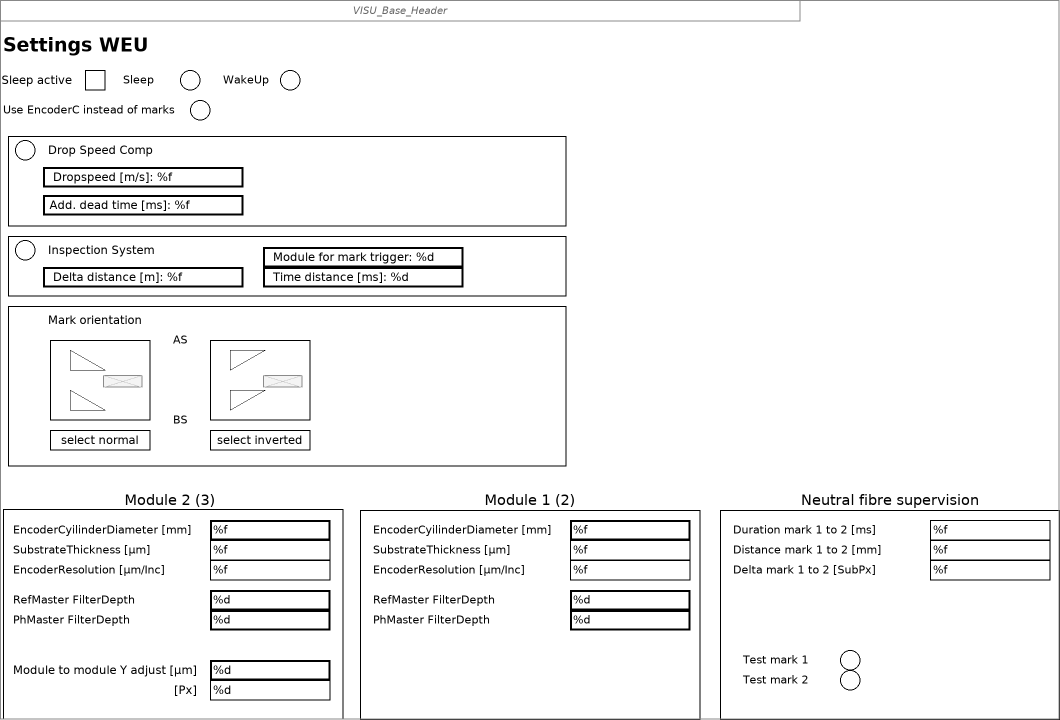
VISUALIZATION VISU_SettingsWeu  // 1060x720
    Rectangle (3,509 340x210)
    Ellipse (190,100 20x20), tooltip "Sim VEncoder"
        toggle PRG_PRINT.bL_EnableEncTrig
    Rectangle (0,100 180x20), "Use EncoderC instead of marks"
    Rectangle (0,30 300x30), "Settings WEU"
    Rectangle (360,510 340x210)
    Label (0,490 340x20), "Module 2 (3)"
    Label (360,490 340x20), "Module 1 (2)"
    Rectangle (10,560 180x20), "EncoderResolution [µm/Inc]"
    Rectangle (210,560 120x20), "%f", text variable: PRG_PRINT.fL_ResolutionEncoder[2]
        OnMouseClick: write the text variable via Default
    Frame (0,0 800x21)
        shows VISU_Base_Header()
    Rectangle (8,136 558x90)
    Ellipse (15,140 20x20), colour toggle: PRG_PRINT.bL_UseSpeedCompensation
        toggle PRG_PRINT.bL_UseSpeedCompensation
    Rectangle (45,140 124x20), "Drop Speed Comp"
    Rectangle (43,167 200x20), "Dropspeed [m/s]: %f", text variable: PRG_PRINT.fL_DropSpeed
        OnMouseDown: write the text variable via Edit
    Rectangle (43,195 200x20), "Add. dead time [ms]: %f", text variable: PRG_PRINT.fL_DropSpeedAddTime
        OnMouseDown: write the text variable via Edit
    Rectangle (370,520 187x20), "EncoderCyilinderDiameter [mm]"
    Rectangle (570,520 120x20), "%f", text variable: PRG_PRINT.lEncoderCylinderDiameter[1]
        OnMouseClick: write the text variable via Default
    RoundedRectangle (85,70 20x20), colour toggle: PRG_MACHINE.sO_SystemCmd.bSleep
    Rectangle (0,70 75x20), "Sleep active"
    Ellipse (180,70 20x20), tooltip "Sim VEncoder"
        tap PRG_MACHINE.bL_SleepVisu
    Rectangle (120,70 55x20), "Sleep"
    Ellipse (280,70 20x20), tooltip "Sim VEncoder"
        tap PRG_MACHINE.bL_WakeUpVisu
    Rectangle (220,70 55x20), "WakeUp"
    Rectangle (210,660 120x20), "%d", text variable: PRG_PRINT.nPrintModuleAdjustY[2]
        OnMouseClick: write the text variable via VisuDialogs.Numpad, min PRG_PRINT.sC_Config_P.lL_PU_GENERALSHIFT_Y_SET_MIN, max PRG_PRINT.sC_Config_P.lL_PU_GENERALSHIFT_Y_SET_MAX
    Rectangle (10,660 190x20), "Module to module Y adjust [µm]"
    Rectangle (370,540 180x20), "SubstrateThickness [µm]"
    Rectangle (570,540 120x20), "%f", text variable: PRG_MACHINE.InEAP_SubstrateThickness
        OnMouseClick: write the text variable via Default
    Rectangle (370,560 180x20), "EncoderResolution [µm/Inc]"
    Rectangle (570,560 120x20), "%f", text variable: PRG_PRINT.fL_ResolutionEncoder[1]
        OnMouseClick: write the text variable via Default
    Rectangle (10,520 187x20), "EncoderCyilinderDiameter [mm]"
    Rectangle (210,520 120x20), "%f", text variable: PRG_PRINT.lEncoderCylinderDiameter[2]
        OnMouseClick: write the text variable via Default
    Rectangle (10,540 180x20), "SubstrateThickness [µm]"
    Rectangle (210,540 120x20), "%f", text variable: PRG_MACHINE.InEAP_SubstrateThickness
        OnMouseClick: write the text variable via Default
    Rectangle (370,590 187x20), "RefMaster FilterDepth"
    Rectangle (570,590 120x20), "%d", text variable: PRG_PRINT.Fb_Ref_Master[1].cI_FilterDepth
        OnMouseClick: write the text variable via Default
    Rectangle (370,610 187x20), "PhMaster FilterDepth"
    Rectangle (570,610 120x20), "%d", text variable: PRG_PRINT.Fb_Ph_Master[1].cI_FilterDepth
        OnMouseClick: write the text variable via Default
    Rectangle (10,590 187x20), "RefMaster FilterDepth"
    Rectangle (210,590 120x20), "%d", text variable: PRG_PRINT.Fb_Ref_Master[2].cI_FilterDepth
        OnMouseClick: write the text variable via Default
    Rectangle (10,610 187x20), "PhMaster FilterDepth"
    Rectangle (210,610 120x20), "%d", text variable: PRG_PRINT.Fb_Ph_Master[2].cI_FilterDepth
        OnMouseClick: write the text variable via Default
    Rectangle (8,236 558x60)
    Ellipse (15,240 20x20), colour toggle: PRG_PRINT.fbInspectionSystemTrigger.bR_Enable
        toggle PRG_PRINT.fbInspectionSystemTrigger.bR_Enable
    Rectangle (45,240 124x20), "Inspection System"
    Rectangle (43,267 200x20), "Delta distance [m]: %f", text variable: PRG_PRINT.fbInspectionSystemTrigger.fR_DeltaDistance, invisible if: Not PRG_PRINT.fbInspectionSystemTrigger._bUsePositionTrigger
        OnMouseDown: write the text variable via VisuDialogs.Numpad, min 0.01
    Rectangle (263,267 200x20), "Time distance [ms]: %d", text variable: PRG_PRINT.fbInspectionSystemTrigger.nR_TimeDistance, invisible if: PRG_PRINT.fbInspectionSystemTrigger._bUsePositionTrigger
        OnMouseDown: write the text variable via VisuDialogs.Numpad, min 10
    Rectangle (263,247 200x20), "Module for mark trigger: %d", text variable: PRG_PRINT.nInspectionSystemMarkIdx, invisible if: PRG_PRINT.fbInspectionSystemTrigger._bUsePositionTrigger
        OnMouseDown: write the text variable via VisuDialogs.Numpad, min 2, max 3
    Rectangle (210,680 120x20), "%d", text variable: PRG_PRINT._nPrintModuleAdjustY[2]
    Rectangle (10,680 190x20), "[Px]"
    Rectangle (720,510 340x210)
    Label (720,490 340x20), "Neutral fibre supervision"
    Rectangle (730,520 180x20), "Duration mark 1 to 2 [ms]"
    Rectangle (930,520 120x20), "%f", text variable: PRG_PRINT.fbNeutralFibreDetermine.fL_DurationMark01to02 / 1000
    Rectangle (730,540 180x20), "Distance mark 1 to 2 [mm]"
    Rectangle (930,540 120x20), "%f", text variable: PRG_PRINT.fbNeutralFibreDetermine.fL_LengthMark01to02
        OnMouseClick: write the text variable via Default
    Rectangle (730,560 180x20), "Delta mark 1 to 2 [SubPx]"
    Rectangle (930,560 120x20), "%f", text variable: PRG_PRINT.fbNeutralFibreDetermine.nL_DeltaMark01to02
        OnMouseClick: write the text variable via Default
    Ellipse (840,650 20x20), tooltip "Sim VEncoder"
        tap PRG_PRINT.fbNeutralFibreDetermine.bIKp_MarkTrigger01
    Rectangle (740,650 100x20), "Test mark 1"
    Ellipse (840,670 20x20), tooltip "Sim VEncoder"
        tap PRG_PRINT.fbNeutralFibreDetermine.bIKp_MarkTrigger02
    Rectangle (740,670 100x20), "Test mark 2"
    Rectangle (8,306 558x160)
    Rectangle (45,310 124x20), "Mark orientation"
    Rectangle (50,340 100x80)
    Polygon (70,350) (70,370) (105,370)
    Polygon (70,390) (70,410) (105,410)
    Image (103,375 39x12), image: VisuSymbols.Symbols.ArrowBoldLeft
    Rectangle (170,330 25x20), "AS"
    Rectangle (170,410 25x20), "BS"
    Rectangle (210,340 100x80)
    Polygon (230,350) (230,370) (265,350)
    Polygon (230,390) (230,410) (265,390)
    Image (263,375 39x12), image: VisuSymbols.Symbols.ArrowBoldLeft
    RoundedRectangle (50,430 100x20), "select normal", colour toggle: NOT PRG_PRINT.bMarksInverted
        tap PRG_PRINT.fbRTrigMarkSelectNormal.CLK
    RoundedRectangle (210,430 100x20), "select inverted", colour toggle: PRG_PRINT.bMarksInverted
        tap PRG_PRINT.fbRTrigMarkSelectInverted.CLK
END_VISUALIZATION

(* stored: Version 1.1.0.1, ProductVersion 3.1.4024.9
   Visu VISU_SettingsWeu: Id {e4f4fc09-bceb-41cf-b9fa-99666ff6f01f} *)
